Staubli VAL3: VALCLEAN.pjx

--- VALCLEAN.pjx ---
Parameters version=s7.8 stackSize=50000 millimeterUnit=true
Program file=kill.pgx
Program file=start.pgx
Program file=stop.pgx
Data file=VALCLEAN.dtx
Library alias=kernel path=Disk://kernel/kernel.pjx autoload=true password=

--- VALCLEAN.dtx ---


--- start.pgx ---
public program start()
  local num i
  local num l_nKey
  local string l_sMessage
begin
  // call the start
  taskCreate "KERNEL",100,kernel:start()
end

--- kill.pgx ---
public program kill()
  local string l_sMessage
begin
  call kernel:_kill()
end

--- stop.pgx ---
program stop()
begin
  //
  // QUIT KERNEL
  //
  call kernel:stop()
  cls()
end
